FUNCTION MF_Sigmoidal : REAL
VAR_INPUT
	x,a,c:REAL;
END_VAR
VAR
	divisor: REAL;
END_VAR

VAR_OUTPUT
	error: BOOL;
END_VAR

divisor:=1+LREAL_TO_REAL(EXP(-a*(x-c)));
IF divisor<>0 THEN	
	MF_Sigmoidal:=1/divisor;
	ELSE error:=TRUE;
END_IF;

END_FUNCTION

(* stored: Version 1.1.0.1, ProductVersion 3.1.4024.6
   POU MF_Sigmoidal: Id {337fabf1-c179-4028-aa23-1f9e7b3c965e}, SpecialFunc None *)
